// TIA Portal V19 export
FUNCTION "CallCmMotor_1" : Void   // FC3, LAD
{ S7_Optimized_Access := 'TRUE' }
// stored: SetENOAutomatically false
BEGIN

NETWORK
TITLE = FT00P01- Interlock and permissive for Motor block
//------------Interlock Status ---------------------
      A     "AlwaysTRUE";
      =     "@DBCmMotor".FT00P01.InterlockStatus[1];
      A     "AlwaysTRUE";
      =     "@DBCmMotor".FT00P01.InterlockStatus[2];
      A     "AlwaysTRUE";
      =     "@DBCmMotor".FT00P01.InterlockStatus[3];
      A     "AlwaysTRUE";
      =     "@DBCmMotor".FT00P01.InterlockStatus[4];
      A     "AlwaysTRUE";
      =     "@DBCmMotor".FT00P01.InterlockStatus[5];
      A     "AlwaysTRUE";
      =     "@DBCmMotor".FT00P01.InterlockStatus[6];
      A     "AlwaysTRUE";
      =     "@DBCmMotor".FT00P01.InterlockStatus[7];
      A     "AlwaysTRUE";
      =     "@DBCmMotor".FT00P01.InterlockStatus[8];
      A     "AlwaysTRUE";
      =     "@DBCmMotor".FT00P01.InterlockStatus[9];
      A     "AlwaysTRUE";
      =     "@DBCmMotor".FT00P01.InterlockStatus[10];
      A     "AlwaysTRUE";
      =     "@DBCmMotor".FT00P01.InterlockStatus[11];
      A     "AlwaysTRUE";
      =     "@DBCmMotor".FT00P01.InterlockStatus[12];
      A     "AlwaysTRUE";
      =     "@DBCmMotor".FT00P01.InterlockStatus[13];
      A     "AlwaysTRUE";
      =     "@DBCmMotor".FT00P01.InterlockStatus[14];
      A     "AlwaysTRUE";
      =     "@DBCmMotor".FT00P01.InterlockStatus[15];
      A     "AlwaysTRUE";
      =     "@DBCmMotor".FT00P01.InterlockStatus[16];



//-----------Persmissive Status ---------------------

      A     "AlwaysTRUE";
      =     "@DBCmMotor".FT00P01.PermissiveStatus[1];
      A     "AlwaysTRUE";
      =     "@DBCmMotor".FT00P01.PermissiveStatus[2];
      A     "AlwaysTRUE";
      =     "@DBCmMotor".FT00P01.PermissiveStatus[3];
      A     "AlwaysTRUE";
      =     "@DBCmMotor".FT00P01.PermissiveStatus[4];
      A     "AlwaysTRUE";
      =     "@DBCmMotor".FT00P01.PermissiveStatus[5];
      A     "AlwaysTRUE";
      =     "@DBCmMotor".FT00P01.PermissiveStatus[6];
      A     "AlwaysTRUE";
      =     "@DBCmMotor".FT00P01.PermissiveStatus[7];
      A     "AlwaysTRUE";
      =     "@DBCmMotor".FT00P01.PermissiveStatus[8];
      A     "AlwaysTRUE";
      =     "@DBCmMotor".FT00P01.PermissiveStatus[9];
      A     "AlwaysTRUE";
      =     "@DBCmMotor".FT00P01.PermissiveStatus[10];
      A     "AlwaysTRUE";
      =     "@DBCmMotor".FT00P01.PermissiveStatus[11];
      A     "AlwaysTRUE";
      =     "@DBCmMotor".FT00P01.PermissiveStatus[12];
      A     "AlwaysTRUE";
      =     "@DBCmMotor".FT00P01.PermissiveStatus[13];
      A     "AlwaysTRUE";
      =     "@DBCmMotor".FT00P01.PermissiveStatus[14];
      A     "AlwaysTRUE";
      =     "@DBCmMotor".FT00P01.PermissiveStatus[15];
      A     "AlwaysTRUE";
      =     "@DBCmMotor".FT00P01.PermissiveStatus[16];



NETWORK
TITLE = FT00P01
// CALL of CM_Motor
      AN    "FT00P01_TRIP";
      =     "FT00P01_TRIP_BIT";

      CALL  "@CmMotor"
      ( i_Remote             := True,
        i_RunFb              := "FT00P01_RUN",
        i_TrippedFb          := "FT00P01_TRIP",
        i_Inhibit            := True,
        i_EStop              := "@DBCmDi".Estop.Status.Active,
        FeatureITripPolarity := "FALSE",
        FirstScanBit         := "FirstScan",
        OneSec               := "OSP",
        SimOn                := "@DBCmMotor".FT00P01.Command.SimOn,
        SimOff               := "@DBCmMotor".FT00P01.Command.SimOff,
        CommonReset          := "@DBCmMotor".FT00P01.Command.LocalFaultReset,
        HooterReset          := "DbHooter".Hooter_Reset,
        AutoReqMode          := "@DBCmMotor".FT00P01.Command.AutoModeReq,
        DCSOperation         := "Loc_Rem_Ctrl",
        q_On                 := "FT00P01_CMD",
        CM                   := "@DBCmMotor".FT00P01
      );



END_FUNCTION
